(* IEC 61131-3 sources: learning-path/07_unit_testing/exercises/solutions/1_starting_tests_solution, 1 file *)

(* ---- test.st ---- *)
USING AxUnit.Assert;
USING Numbers;

NAMESPACE Test
    {Test}
    FUNCTION EvenNumber
        VAR_TEMP
            result : BOOL;
        END_VAR

        result := NumberIsEven(2);
        Equal(actual := result, expected := TRUE);

        result := NumberIsEven(5);
        Equal(actual := result, expected := FALSE);
    END_FUNCTION
END_NAMESPACE
